FUNCTION FindMinMax 
VAR_INPUT
	aWeight : ARRAY[1..20] OF REAL;
END_VAR
VAR_IN_OUT
    minWeight : REAL;
	maxWeight : REAL;
END_VAR
VAR
	i : INT;
	
END_VAR

 minWeight := aWeight[1];
maxWeight := aWeight[1];

     FOR i:=1 TO 20 DO
		 IF aWeight[i]>maxWeight THEN
			 maxWeight := aWeight[i];
		 END_IF
		 
		 IF aWeight[i]<minWeight THEN
			 minWeight := aWeight[i];
		 END_IF
		 
	 END_FOR

END_FUNCTION

(* stored: Version 1.1.0.1, ProductVersion 3.1.4024.16
   POU FindMinMax: Id {ecb9de9b-3a2e-421d-a18e-1116866eb408}, SpecialFunc None *)
